TYPE stDetectionTunelParams :
STRUCT
	rBottleLoad				: REAL;
	rBottleLoadTolerance	: REAL;
	iConvoyerMaxSpeed		: INT;
	iSpeedingTime			: INT;
	iDropedBottlesLimit		: BYTE;
	bWeightCheck			: BOOL;
	bCognexEnable			: BOOL;
	bOrangeExpected			: BOOL;	//Input 2
	bGreenExpected			: BOOL; //Input 1
	rConvoyerSpeed			: REAL;
	iForceStabilTime		: INT;
	iStartWaitTime			: INT;
	iDetectionWaitTime		: INT;
	iFilterStabilizationTime	: UINT := 250;
	bAutoTaringEnable		: BOOL := FALSE;
END_STRUCT
END_TYPE

(* stored: Version 1.1.0.1, ProductVersion 3.1.4024.13
   DUT stDetectionTunelParams: Id {57160bfc-a13e-4ee6-ac09-e2790bc80290} *)
